TYPE eXMLState :
(
	
	eWait,
eResetWrite, 
eWriteData, 
eResetRead, 
eReadData
);
END_TYPE

(* stored: Version 1.1.0.1, ProductVersion 3.1.0.38
   DUT eXMLState: Id {c9357433-fb9d-440a-9985-38682bdb1d74} *)
